// TIA Portal V19 export
TYPE "lexchangetray_typeUnEmn_toHandlingXyzRecieve"
// Type: lexchangetray_typehandlingXyzEm_toConstraintRollerReq
// Type: lexchangetray_typehandlingXyzEm_toConstraintRollerFeedback
// stored: Access Published
   STRUCT
      feedback { S7_SetPoint := 'True'} : "lexchangetray_typehandlingXyzEm_toConstraintRollerFeedback";
      req { S7_SetPoint := 'True'} : "lexchangetray_typehandlingXyzEm_toConstraintRollerReq";
   END_STRUCT;
END_TYPE
